SUBAPPLICATION mapping_Uebung_034b (* LONG_PRESS_HOLD-Eingang auf PWM Ausgang *)
  (* Standard: 61499-2; Description: Copyright (c) 2023 Meisterschulen am Ostbahnhof This program and the accompanying materials are made available under the terms of the Eclipse Public License 2.0 which is available at https://www.eclipse.org/legal/epl-2.0/ SPDX-License-Identifier: EPL-2.0 *)
  (* Version 1.0, 2023-10-23, Franz Höpfinger, Meisterschulen am Ostbahnhof *)
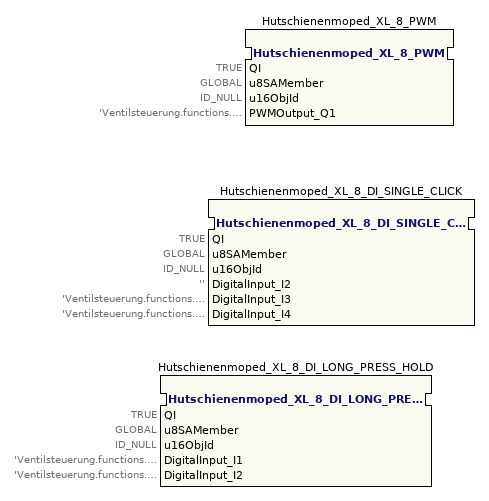
  FBS
    Hutschienenmoped_XL_8_PWM : Hutschienenmoped_XL_8_PWM(QI := TRUE, u8SAMember := GLOBAL, u16ObjId := ID_NULL, PWMOutput_Q1 := 'Ventilsteuerung.functions.PWMOutput_Q1');
    Hutschienenmoped_XL_8_DI_SINGLE_CLICK : Hutschienenmoped_XL_8_DI_SINGLE_CLICK(QI := TRUE, u8SAMember := GLOBAL, u16ObjId := ID_NULL, DigitalInput_I2 := '', DigitalInput_I3 := 'Ventilsteuerung.functions.IE_STOP', DigitalInput_I4 := 'Ventilsteuerung.functions.IE_FULL');
    Hutschienenmoped_XL_8_DI_LONG_PRESS_HOLD : Hutschienenmoped_XL_8_DI_LONG_PRESS_HOLD(QI := TRUE, u8SAMember := GLOBAL, u16ObjId := ID_NULL, DigitalInput_I1 := 'Ventilsteuerung.functions.IE_SPEED_UP', DigitalInput_I2 := 'Ventilsteuerung.functions.IE_SPEED_DOWN');
  END_FBS
END_SUBAPPLICATION
